(* CODESYS project CODESYS-Minimum-Test

Project tree, tasks and I/O mapping:
  Device : CODESYS Control for Raspberry Pi 64 SL, CODESYS, order no. 2302000009, version 4.15.0.0
    application Application
      libraries: Standard, 3.5.18.0 (System)
      task MainTask (cyclic, interval t#4ms, priority 1) calls PLC_PRG
      program PLC_PRG [ST]
    Camera device
      <Leer>
    GPIOs_A_B : GPIOs A/B, CODESYS, version 4.15.0.0
        unmapped channels: digital inputs (GPIO0..GPIO31), digital outputs (GPIO0..GPIO31)
    I²C
    Onewire
    SoftMotion General Axis Pool
    SPI
*)

// Device/Application/PLC_PRG
PROGRAM PLC_PRG
VAR
	i: INT;
END_VAR


i := i+1;

END_PROGRAM
